INTERFACE I_Job  EXTENDS __SYSTEM.IQueryInterface

(*abort method

*)
METHOD abort : BOOL // Return TRUE if finish.
VAR_INPUT
END_VAR
END_METHOD

PROPERTY busy : BOOL
GET
END_GET
END_PROPERTY

PROPERTY children : InterfaceContainer // Accesser for interface pointer to child container instance.
GET
END_GET
END_PROPERTY

PROPERTY continuous_mode : bool // Make true if keep executing state after all jobs be finished.
SET
END_SET
END_PROPERTY

METHOD create_container : InterfaceContainer // Make container object onto child.
VAR_INPUT
	container_type : ContainerType; // specify container type
	name: STRING;	// specify future name
END_VAR
END_METHOD

METHOD create_future : InterfaceFuture // Create future dynamically.
VAR_INPUT
	creator : InterfaceTaskCreator; // Specify creator object by which Interface Task Creator implemented.
	future_name: STRING; // Spcfigy future name.
END_VAR
END_METHOD

{attribute 'OPC.UA.DA.Property' := '1'}
{attribute 'monitoring' := 'call'}
{attribute 'OPC.UA.DA.Description' := 'Current state of this executor object.'}
PROPERTY current_state : E_FutureExecutionState // Get current job state
GET
END_GET
END_PROPERTY

PROPERTY current_timestamp : POINTER TO T_FILETIME64
GET
END_GET
SET
END_SET
END_PROPERTY

PROPERTY done : BOOL // Present true if process be finished.
GET
END_GET
END_PROPERTY

METHOD error_reset : BOOL
VAR_INPUT
END_VAR
END_METHOD

METHOD execute : BOOL // Execute future process and return TRUE if all task are finished.
END_METHOD

PROPERTY future : InterfaceFuture // Set future instance direct.
GET
END_GET
SET
END_SET
END_PROPERTY

PROPERTY future_creator : InterfaceTaskCreator // Set creator instance.
SET
END_SET
END_PROPERTY

METHOD get_job_info : BOOL
VAR_INPUT
	title		: T_MaxString;
	observable 	: I_Observable;
	recursive	: BOOL := FALSE;
END_VAR
END_METHOD

PROPERTY id : T_MaxString // Get job id.
GET
END_GET
SET
END_SET
END_PROPERTY

METHOD init : BOOL // Return TRUE if finish.
VAR_INPUT
END_VAR
END_METHOD

PROPERTY job_event_reporter : I_JobInfo
GET
END_GET
SET
END_SET
END_PROPERTY

PROPERTY last_state : E_FutureExecutionState
GET
END_GET
END_PROPERTY

PROPERTY lid : T_MaxString
GET
END_GET
END_PROPERTY

PROPERTY namespace : T_MaxString
GET
END_GET
END_PROPERTY

PROPERTY nErrorID : HRESULT // Present error code when each process,init(), execute(), quit() are finished. '0' represent normal condition without any errors.
GET
END_GET
END_PROPERTY

PROPERTY parent_executor : I_Job
GET
END_GET
SET
END_SET
END_PROPERTY

PROPERTY persistent_job : BOOL
GET
END_GET
SET
END_SET
END_PROPERTY

METHOD quit : BOOL // Return TRUE if finish.
VAR_INPUT
END_VAR
END_METHOD

PROPERTY ready : BOOL
GET
END_GET
END_PROPERTY

METHOD reset : BOOL // Return TRUE if finish.
VAR_INPUT
	deep : BOOL := FALSE;
END_VAR
END_METHOD

METHOD resume : BOOL
END_METHOD

METHOD start : BOOL
END_METHOD

PROPERTY uid : T_MaxString
GET
END_GET
END_PROPERTY

PROPERTY upstream_aborting : BOOL
GET
END_GET
SET
END_SET
END_PROPERTY

END_INTERFACE

(* stored: Version 1.1.0.1, ProductVersion 3.1.4026.13
   Itf I_Job: Id {c241c129-013a-48a7-8f50-a46604fd73e8}
   Method abort: Id {ba384c68-144d-4364-9ff2-dddd491ec19b}
   Property busy: Id {0a37f028-1504-4cb9-b1b7-53bde72f8218}
   Get Get: Id {3fc6c967-5220-403e-87b7-749035c24bde}
   Property children: Id {22f1430e-f0f4-41f2-b46c-84e39d72eef9}
   Get Get: Id {15e6d966-0d98-49a3-b8d2-a7b46a69e496}
   Property continuous_mode: Id {5447b52e-b242-4675-8469-7326885828e2}
   Set Set: Id {a2ab253f-3721-4987-9553-9b003b002196}
   Method create_container: Id {ef3659a9-663f-436e-aba6-183a0f497e09}
   Method create_future: Id {b2304e27-07e6-4812-a102-238f555d4211}
   Property current_state: Id {3bfa10c5-3b1a-417f-a36e-93b29914da62}
   Get Get: Id {96511d7e-81ae-459b-9a47-3a200cb859d4}
   Property current_timestamp: Id {b926ced9-2489-4467-805a-e7d95bed8cdf}
   Get Get: Id {a8d3ca2d-d89a-4442-b154-5f9ccad5ba29}
   Set Set: Id {04885ff6-8be2-40f0-a6f5-2042bf59e436}
   Property done: Id {49aa35c1-9eff-40f2-9175-654e8db9ac55}
   Get Get: Id {45954038-aba4-4ca0-9dca-c851b3710f18}
   Method error_reset: Id {fb5cadc3-27be-41ec-9249-633dbdf2cb4f}
   Method execute: Id {409ed4e0-c300-4f5d-ae79-ae3e1916ca1c}
   Property future: Id {7eb38465-3b0f-45b2-8963-3234ef5b537d}
   Get Get: Id {b2111c34-68f3-4c57-8cbb-f8aca8c3cab9}
   Set Set: Id {2dd1e9c2-d6b2-4b75-aa3e-9b57cc7b06b8}
   Property future_creator: Id {4453c69f-5993-4e32-aa6b-70c0a3524612}
   Set Set: Id {4c5d6441-82c1-43cc-a85e-15d729c30d05}
   Method get_job_info: Id {dcf93f75-a375-4062-b2dd-3955dc6dab77}
   Property id: Id {7e4a5eb7-1da6-498f-b820-0b35913287d7}
   Get Get: Id {cd5b6e57-c851-4790-b895-552dc87d0850}
   Set Set: Id {6956f113-09b2-4acc-bbc2-bf32e24ecb97}
   Method init: Id {d81bf7e0-a419-45a2-a8da-d29900ce51e8}
   Property job_event_reporter: Id {86842a8e-fd31-4199-9e8a-898c1d1cd9cd}
   Get Get: Id {99052aa6-8cde-4c37-b866-4701a11893cf}
   Set Set: Id {f32ae562-a901-42d1-862f-6e9bedd113ca}
   Property last_state: Id {c0d32629-3739-44a6-a76a-562079ce9773}
   Get Get: Id {516dfae1-5a01-4cc5-bfd0-d6e15004cff0}
   Property lid: Id {630d76a2-75c7-40d8-ad23-f5f0e325fe2e}
   Get Get: Id {a0799991-7d39-4da9-8d77-69af7e855799}
   Property namespace: Id {3fd49687-b433-46f1-b4e3-da6564312bf5}
   Get Get: Id {a073b4a6-1d91-4c1f-b46b-586a3d540fad}
   Property nErrorID: Id {587d3aee-efb4-44d2-8930-476a7f1c0617}
   Get Get: Id {a3d3ab3d-9d97-4c08-af3c-1d49e2061134}
   Property parent_executor: Id {afe0c2b8-f9fa-47b0-90ee-38d73ecdf14f}
   Get Get: Id {1ff8349f-c5a4-4d15-9d8a-dec4e14daa55}
   Set Set: Id {3598cf4f-5a6f-40b3-9da7-3117baa0a6ef}
   Property persistent_job: Id {4e7348c0-cfaa-4896-a661-211f010820db}
   Get Get: Id {bb9fa261-ba47-4735-8f86-0557267d8ac3}
   Set Set: Id {f2ea2f19-1746-4bf2-955a-0d91fb6a9b2a}
   Method quit: Id {31796530-93ca-4ab0-8e11-4aa4e570a94a}
   Property ready: Id {6e637a5d-a326-4126-bf27-305dae1a03d1}
   Get Get: Id {d20fe530-72fb-41ed-8821-b41c52e366ff}
   Method reset: Id {834f043c-6964-4495-9c44-b9225b356eb2}
   Method resume: Id {7b0c46e2-dfa2-44c4-83df-ea3de905fb2f}
   Method start: Id {85cad871-c4a3-42b3-ac51-d1ea4715df17}
   Property uid: Id {116d0832-62fe-4e90-8de4-5a2758b3baec}
   Get Get: Id {6371e964-9ef9-4dae-ab0f-1650739a8d2b}
   Property upstream_aborting: Id {a7842f50-8df5-46f1-ab16-88ebb4c8aa74}
   Get Get: Id {13e86aa0-64b7-4dbf-a816-21154bcabe6a}
   Set Set: Id {8c26813a-2b94-4eff-91e3-a173456bd1af} *)
